// TIA Portal V17 export
// export: Created 2024-08-29T18:23:50.3233838Z, ExportSetting WithDefaults, DisplayName Totally Integrated Automation Portal, DisplayVersion V17 Update 7, DisplayName TIA Portal Openness, DisplayVersion V17 Update 7, DisplayName TIA Portal Version Control Interface, DisplayVersion V17, DisplayName SINAMICS Startdrive Advanced, DisplayVersion V17 SP2, DisplayName SINAMICS Startdrive G110M, G120, G120C, G120D, G120P, G115D, DisplayVersion V17 SP2, DisplayName SINAMICS Startdrive G130, G150, S120, S150, SINAMICS MV, S210, DisplayVersion V17 SP2, DisplayName STEP 7 Professional, DisplayVersion V17 Update 7, DisplayName STEP 7 Safety, DisplayVersion V17 Update 6, DisplayName WinCC Advanced / Unified PC, DisplayVersion V17 Update 7
VAR_GLOBAL   // PLC tag table "alarmMemory"
   alarm0 AT %MW100 : Int;   // alarm number
   alarm1 AT %MW102 : Int;   // alarm number
   alarm2 AT %MW104 : Int;
   retIolink AT %MW108 : Int;
   retManifold AT %MW112 : Int;
   retEuchner AT %MW106 : Int;
   retIolink2 AT %MW110 : Int;
   QuitarErrorEscaner AT %MW6 : Word;
   bypass4 AT %M2.3 : Bool;
   bypass5 AT %M2.4 : Bool;
   retPrinter AT %MW114 : Int;
   reProfinetIO1 AT %MW116 : Int;
   reProfinetIO2 AT %MW118 : Int;
   reProfinetIO3 AT %MW120 : Int;
END_VAR
